FUNCTION_BLOCK AutimaticMotion
VAR_INPUT
END_VAR
VAR_OUTPUT
END_VAR
VAR
END_VAR

// NETWORK 1

END_FUNCTION_BLOCK

(* stored: Version 1.1.0.1, ProductVersion 3.1.4024.4
   POU AutimaticMotion: Id {36d09308-31a3-425a-b7f2-0c629caa461b}, SpecialFunc None *)
